TYPE EM_TransportCanSupply2_PAR :
STRUCT
END_STRUCT
END_TYPE

(* stored: Version 1.1.0.1, ProductVersion 3.1.4024.12
   DUT EM_TransportCanSupply2_PAR: Id {6c27e812-3b4f-4f00-96b2-ee83f9fc2841} *)
